ABB RAPID module: CalibData.modx

MODULE CalibData
    PERS tooldata tool2:=[TRUE,[[-53.619,0.072,146.999],[1,0,0,0]],[1,[-56.457,-4.303,139.607],[1,0,0,0],0,0,0]];
ENDMODULE
